// TIA Portal V16 export
// export: Created 2021-08-10T11:53:40.4139441Z, ExportSetting WithDefaults, WithReadOnly, DisplayName Totally Integrated Automation Portal, DisplayVersion V16, DisplayName TIA Portal Version Control Interface, DisplayVersion V16, DisplayName TIA Portal Openness, DisplayVersion V16, DisplayName TIA Portal Teamcenter Gateway, DisplayVersion V16, DisplayName SINAMICS Startdrive Advanced, DisplayVersion V16, DisplayName SINAMICS Startdrive G130, G150, S120, S150, SINAMICS MV, S210, DisplayVersion V16, DisplayName SINAMICS Startdrive G110M, G120, G120C, G120D, G120P, DisplayVersion V16, DisplayName STEP 7 Professional, DisplayVersion V16, DisplayName STEP 7 Safety, DisplayVersion V16, DisplayName WinCC Unified SCADA Engineering System, DisplayVersion V16
FUNCTION_BLOCK "fbValve_Solenoid"   // FB110, FBD
TITLE = Controls a double- or single-acting valve
{ S7_Optimized_Access := 'TRUE' }
VERSION : 0.1
// stored: AutoNumber false, CodeModifiedDate 2021-08-10T11:52:58.0273326Z, CompileDate 2021-08-10T11:53:23.0999729Z, CreationDate 2020-02-26T07:34:28.9567791Z, DownloadWithoutReinit false, HandleErrorsWithinBlock false, InterfaceModifiedDate 2019-07-17T06:42:37.7805928Z, IsConsistent true, IsIECCheckEnabled false, IsKnowHowProtected false, ISMultiInstanceCapable true, IsRetainMemResEnabled false, IsWriteProtected false, LibraryConformanceStatus Warning: The object contains access to global PLC constants., LibraryType fbValve_Solenoid V 3.0.6 in test, LibraryTypeVersionGuid 0a9fd967-cd2b-46e1-afc3-82055bb762c7, MemoryReserve 100, ModifiedDate 2021-08-10T11:52:58.0273326Z, ParameterModified 2019-07-17T06:42:37.7805928Z, PLCSimAdvancedSupport true, SetENOAutomatically false, StructureModified 2019-07-17T06:42:37.7805928Z, UDAEnableTagReadback false
   VAR_INPUT
      tInTimeout { ExternalAccessible := 'False'; ExternalVisible := 'False'; ExternalWritable := 'False'} : Time;   // Timeout time for an actuator's feedback to activate before giving a fault
      iInMode { ExternalAccessible := 'False'; ExternalVisible := 'False'; ExternalWritable := 'False'} : Int;   // Mode Selection
      bInEstop { ExternalAccessible := 'False'; ExternalVisible := 'False'; ExternalWritable := 'False'} : Bool;   // Estop
      bInSignalHome { ExternalAccessible := 'False'; ExternalVisible := 'False'; ExternalWritable := 'False'} : Bool;   // Home position feedback
      bInSignalWork { ExternalAccessible := 'False'; ExternalVisible := 'False'; ExternalWritable := 'False'} : Bool;   // Work position feedback
      bInEnable { ExternalAccessible := 'False'; ExternalVisible := 'False'; ExternalWritable := 'False'} : Bool;   // Home and Work Enabled
      bInCommandWork { ExternalAccessible := 'False'; ExternalVisible := 'False'; ExternalWritable := 'False'} : Bool;   // Move to work position in automatic mode
      bInResetError { ExternalAccessible := 'False'; ExternalVisible := 'False'; ExternalWritable := 'False'} : Bool;   // Reset Error
      bInSimulate { ExternalAccessible := 'False'; ExternalVisible := 'False'; ExternalWritable := 'False'} : Bool;   // Activate device simulation
   END_VAR
   VAR_OUTPUT
      bOutCommandHome { ExternalAccessible := 'False'; ExternalVisible := 'False'; ExternalWritable := 'False'} : Bool;   // Home position command
      bOutCommandWork { ExternalAccessible := 'False'; ExternalVisible := 'False'; ExternalWritable := 'False'} : Bool;   // Work position command
      bOutActiveHome { ExternalAccessible := 'False'; ExternalVisible := 'False'; ExternalWritable := 'False'} : Bool;   // Valve is in home position
      bOutActiveWork { ExternalAccessible := 'False'; ExternalVisible := 'False'; ExternalWritable := 'False'} : Bool;   // Valve is in work position
      bOutAuto { ExternalAccessible := 'False'; ExternalVisible := 'False'; ExternalWritable := 'False'} : Bool;   // Block in auto mode
      bOutError { ExternalAccessible := 'False'; ExternalVisible := 'False'; ExternalWritable := 'False'} : Bool;   // Error exists
      ERROR_Valve { ExternalAccessible := 'False'; ExternalVisible := 'False'; ExternalWritable := 'False'} : "udtError_Valve";   // Valve error structure
   END_VAR
   VAR_IN_OUT
      HMI_ValveControl : "udtHMI_ValveControl";   // HMI valve control
   END_VAR
   VAR
      ErrorScroller { ExternalAccessible := 'False'; ExternalVisible := 'False'; ExternalWritable := 'False'; S7_SetPoint := 'True'} : "fbErrorScroller";   // Sub-block to handle error scroller
      TON_TimeOut { ExternalAccessible := 'False'; ExternalVisible := 'False'; ExternalWritable := 'False'; S7_SetPoint := 'True'} : TON_TIME;   // Timer for Error Timeout
      iLastMode { ExternalAccessible := 'False'; ExternalVisible := 'False'; ExternalWritable := 'False'} : Int;   // Last mode code
      bNewMode { ExternalAccessible := 'False'; ExternalVisible := 'False'; ExternalWritable := 'False'} : Bool;   // New mode selected
      bEnableHome { ExternalAccessible := 'False'; ExternalVisible := 'False'; ExternalWritable := 'False'} : Bool;   // Home position enabled
      bEnableWork { ExternalAccessible := 'False'; ExternalVisible := 'False'; ExternalWritable := 'False'} : Bool;   // Work position enabled
      bAutoMode { ExternalAccessible := 'False'; ExternalVisible := 'False'; ExternalWritable := 'False'} : Bool;   // Auto Mode is active
      bManualMode { ExternalAccessible := 'False'; ExternalVisible := 'False'; ExternalWritable := 'False'} : Bool;   // Manual Mode is active
      bReset { ExternalAccessible := 'False'; ExternalVisible := 'False'; ExternalWritable := 'False'} : Bool;
      bTON_TimeOut { ExternalAccessible := 'False'; ExternalVisible := 'False'; ExternalWritable := 'False'} : Bool;
      bPB_Home { ExternalAccessible := 'False'; ExternalVisible := 'False'; ExternalWritable := 'False'} : Bool;
      bPB_Work { ExternalAccessible := 'False'; ExternalVisible := 'False'; ExternalWritable := 'False'} : Bool;
      bPB_ResetError { ExternalAccessible := 'False'; ExternalVisible := 'False'; ExternalWritable := 'False'} : Bool;
   END_VAR
   VAR_TEMP
      tTimeoutElapsed : Time;   // Elapsed time for TON_Timeout
      bTemp : Bool;
   END_VAR
   VAR_TEMP   // added for the SCL form of the ladder/FBD networks
      _w1 : Bool;
      _w2 : Bool;
   END_VAR
BEGIN

REGION Network 1: --------------------------------------------------------- Inputs ------------------------------------------------------------------
END_REGION

REGION Network 2: Read HMI input buttons
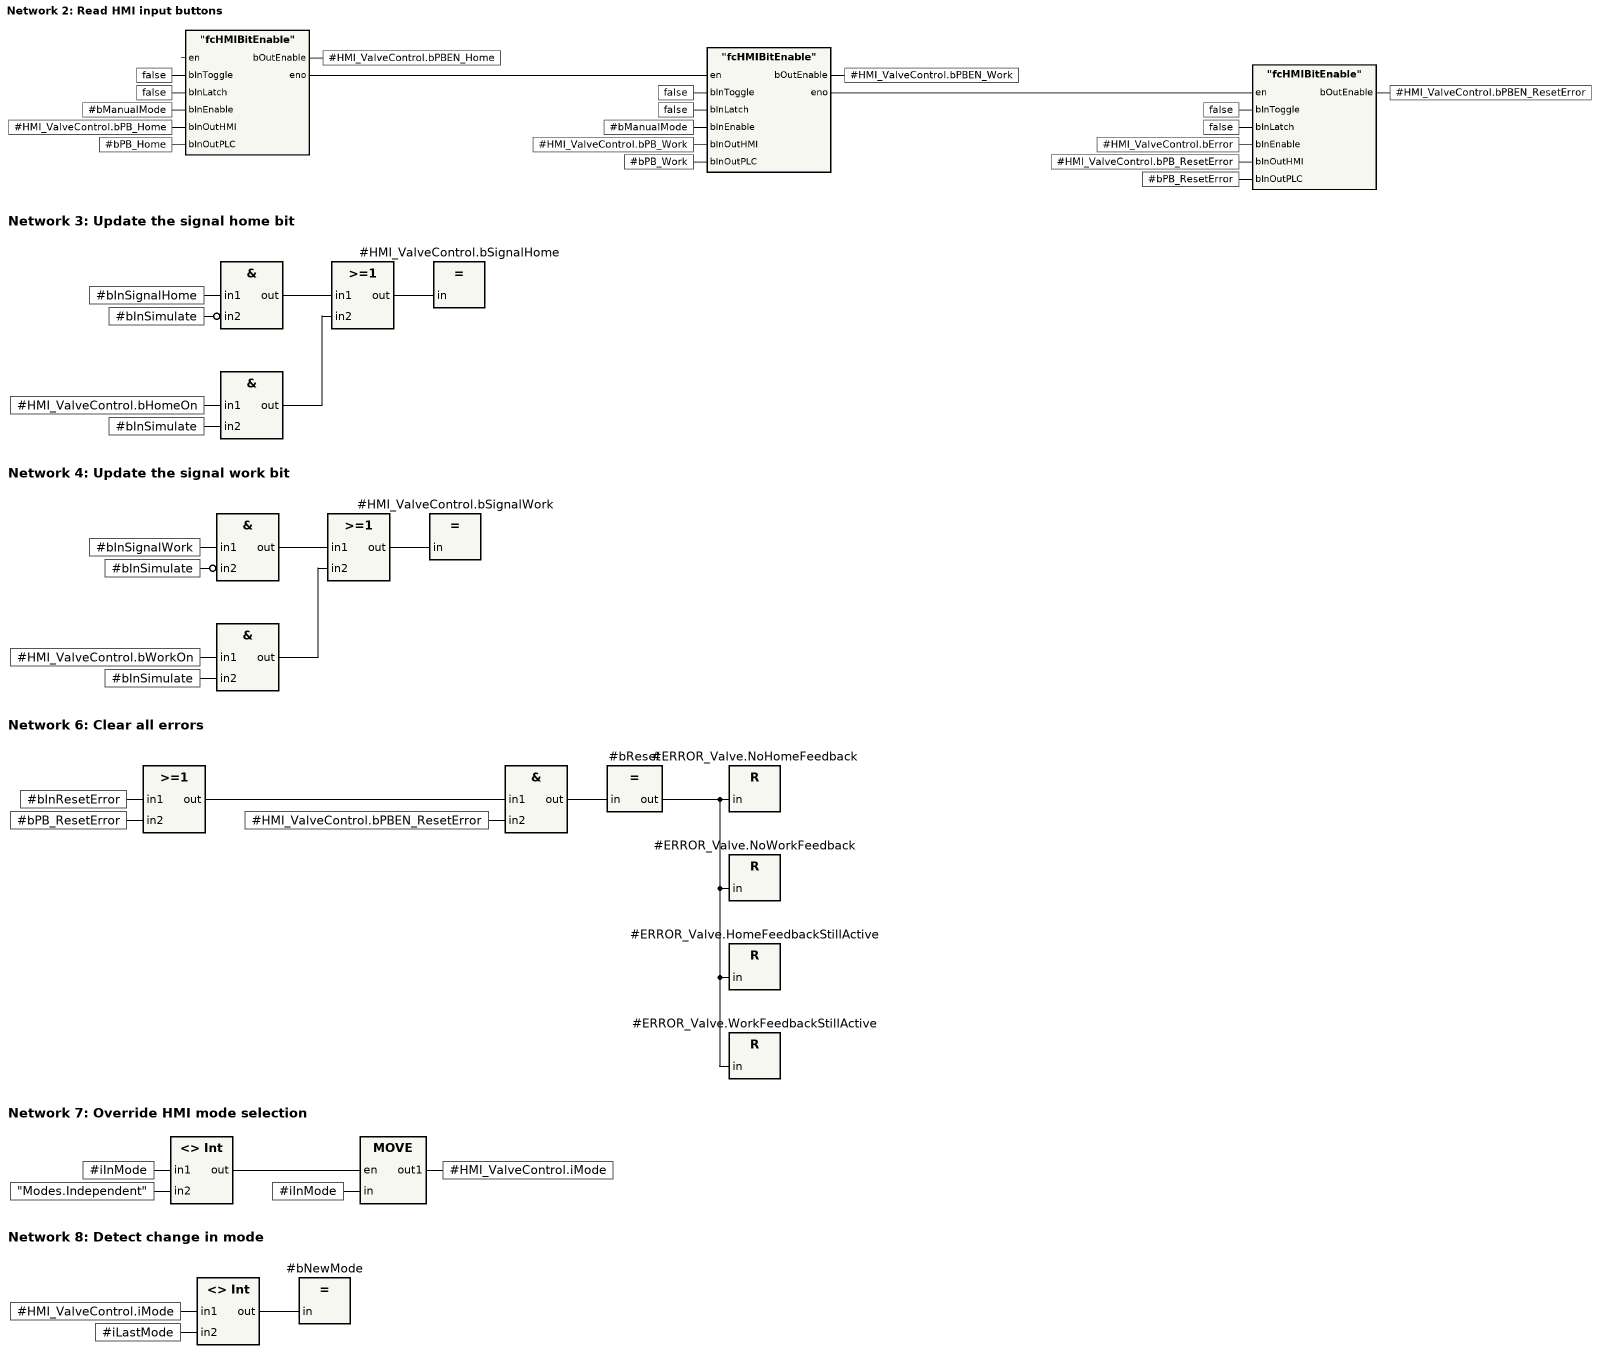
   "fcHMIBitEnable"(bInToggle := false,
                    bInLatch := false,
                    bInEnable := #bManualMode,
                    bInOutHMI := #HMI_ValveControl.bPB_Home,
                    bInOutPLC := #bPB_Home,
                    bOutEnable => #HMI_ValveControl.bPBEN_Home,
                    ENO => #_w1);
   "fcHMIBitEnable"(EN := #_w1,
                    bInToggle := false,
                    bInLatch := false,
                    bInEnable := #bManualMode,
                    bInOutHMI := #HMI_ValveControl.bPB_Work,
                    bInOutPLC := #bPB_Work,
                    bOutEnable => #HMI_ValveControl.bPBEN_Work,
                    ENO => #_w2);
   IF #_w2 THEN
       "fcHMIBitEnable"(bInToggle := false,
                        bInLatch := false,
                        bInEnable := #HMI_ValveControl.bError,
                        bInOutHMI := #HMI_ValveControl.bPB_ResetError,
                        bInOutPLC := #bPB_ResetError,
                        bOutEnable => #HMI_ValveControl.bPBEN_ResetError);
   END_IF;
END_REGION

REGION Network 3: Update the signal home bit
   #HMI_ValveControl.bSignalHome := (#bInSignalHome AND NOT #bInSimulate) OR (#HMI_ValveControl.bHomeOn AND #bInSimulate);
END_REGION

REGION Network 4: Update the signal work bit
   #HMI_ValveControl.bSignalWork := (#bInSignalWork AND NOT #bInSimulate) OR (#HMI_ValveControl.bWorkOn AND #bInSimulate);
END_REGION

REGION Network 5: --------------------------------------------------- Control Logic ------------------------------------------------------------
END_REGION

REGION Network 6: Clear all errors
   #bReset := (#bInResetError OR #bPB_ResetError) AND #HMI_ValveControl.bPBEN_ResetError;
   IF #bReset THEN
       #ERROR_Valve.NoHomeFeedback := FALSE;
       #ERROR_Valve.NoWorkFeedback := FALSE;
       #ERROR_Valve.HomeFeedbackStillActive := FALSE;
       #ERROR_Valve.WorkFeedbackStillActive := FALSE;
   END_IF;
END_REGION

REGION Network 7: Override HMI mode selection
   IF #iInMode <> "Modes.Independent" THEN #HMI_ValveControl.iMode := #iInMode; END_IF;
END_REGION

REGION Network 8: Detect change in mode
   #bNewMode := #HMI_ValveControl.iMode <> #iLastMode;
END_REGION

REGION Network 9: Keep track of last mode
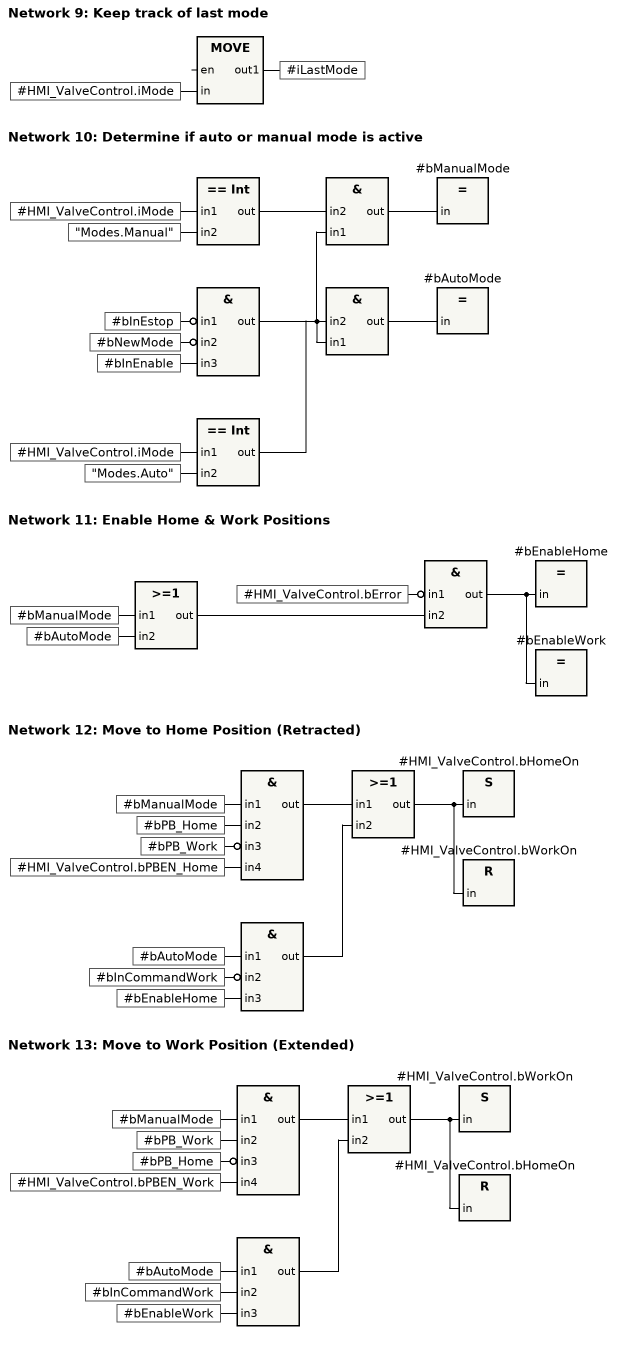
   #iLastMode := #HMI_ValveControl.iMode;
END_REGION

REGION Network 10: Determine if auto or manual mode is active
   #_w1 := NOT #bInEstop AND NOT #bNewMode AND #bInEnable;
   #bManualMode := (#HMI_ValveControl.iMode = "Modes.Manual") AND #_w1;
   #bAutoMode := (#HMI_ValveControl.iMode = "Modes.Auto") AND #_w1;
END_REGION

REGION Network 11: Enable Home & Work Positions
   // IF manual mode AND no estop AND not a new mode AND enabled => 
   // --if no cylinder errors, enable move to Home and Work
   // --enable home and work HMI buttons only in manual mode
   #bEnableHome := NOT #HMI_ValveControl.bError AND (#bManualMode OR #bAutoMode);
   #bEnableWork := #bEnableHome;
END_REGION

REGION Network 12: Move to Home Position (Retracted)
   // IF manual mode and home button is pressed =>
   // --Set close cylinder
   IF (#bManualMode AND #bPB_Home AND NOT #bPB_Work AND #HMI_ValveControl.bPBEN_Home) OR (#bAutoMode AND NOT #bInCommandWork AND #bEnableHome) THEN
       #HMI_ValveControl.bHomeOn := TRUE;
       #HMI_ValveControl.bWorkOn := FALSE;
   END_IF;
END_REGION

REGION Network 13: Move to Work Position (Extended)
   // IF manual mode and work button button is pressed =>
   // --Set open cylinder
   IF (#bManualMode AND #bPB_Work AND NOT #bPB_Home AND #HMI_ValveControl.bPBEN_Work) OR (#bAutoMode AND #bInCommandWork AND #bEnableWork) THEN
       #HMI_ValveControl.bWorkOn := TRUE;
       #HMI_ValveControl.bHomeOn := FALSE;
   END_IF;
END_REGION

REGION Network 14: Reset home on if not enabled
   // IF in auto AND home is not enabled => RESET home command
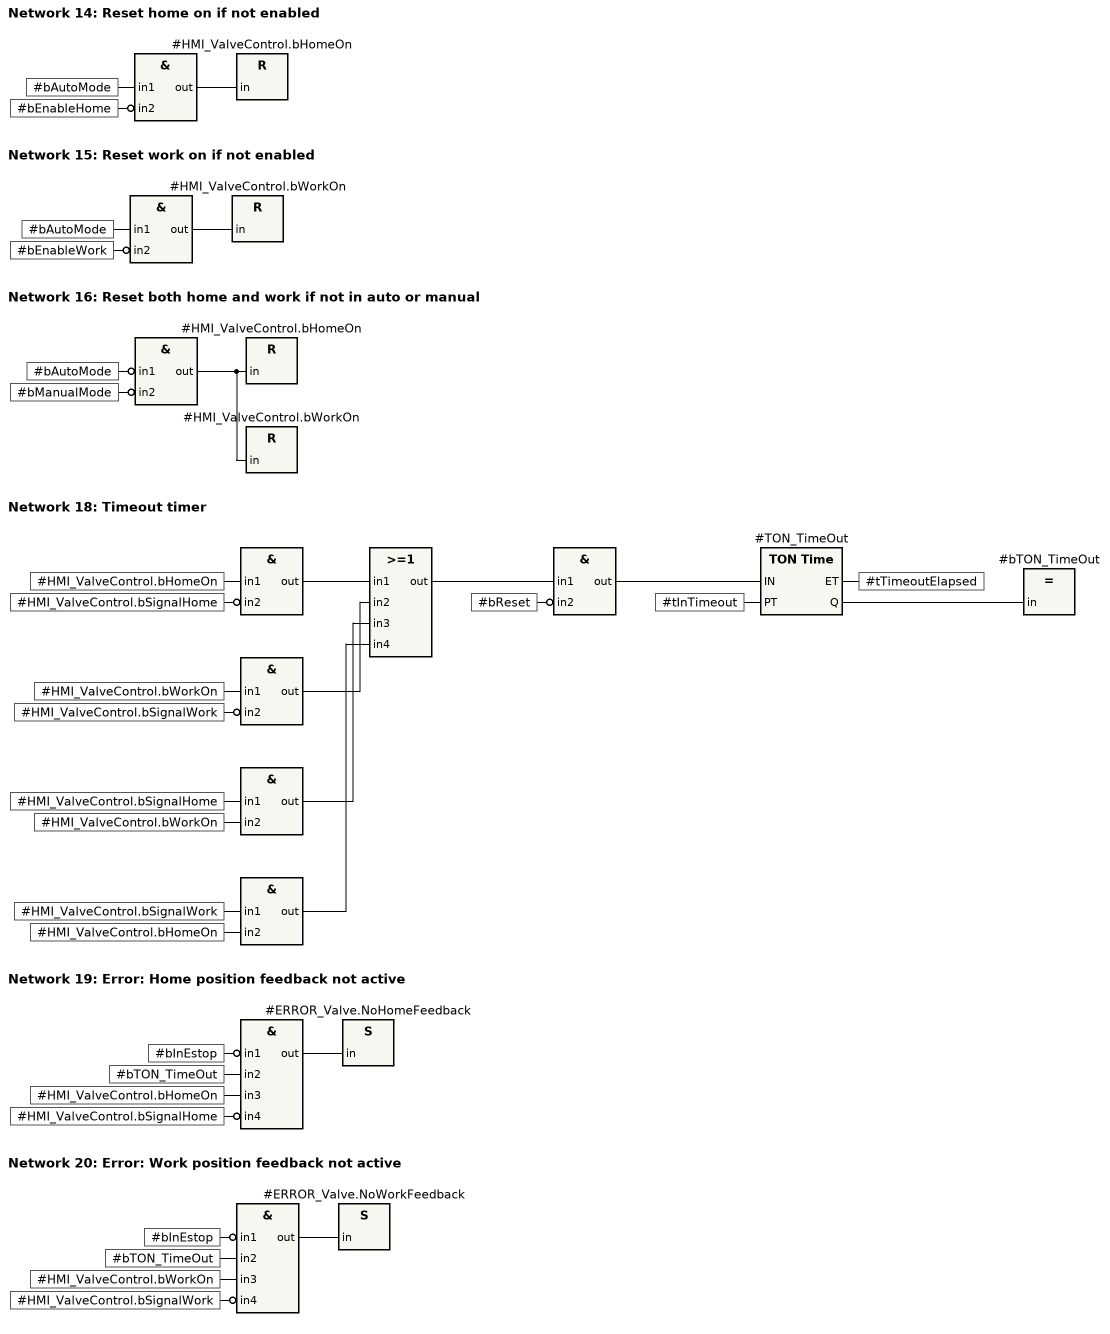
   IF #bAutoMode AND NOT #bEnableHome THEN #HMI_ValveControl.bHomeOn := FALSE; END_IF;
END_REGION

REGION Network 15: Reset work on if not enabled
   // IF in auto AND work is not enabled => RESET work command
   IF #bAutoMode AND NOT #bEnableWork THEN #HMI_ValveControl.bWorkOn := FALSE; END_IF;
END_REGION

REGION Network 16: Reset both home and work if not in auto or manual
   // IF not in auto AND not in manual => RESET home and work commands
   IF NOT #bAutoMode AND NOT #bManualMode THEN
       #HMI_ValveControl.bHomeOn := FALSE;
       #HMI_ValveControl.bWorkOn := FALSE;
   END_IF;
END_REGION

REGION Network 17: --------------------------------------------------------- Errors ------------------------------------------------------------------
END_REGION

REGION Network 18: Timeout timer
   // Time delay for errors
   #TON_TimeOut(IN := ((#HMI_ValveControl.bHomeOn AND NOT #HMI_ValveControl.bSignalHome) OR (#HMI_ValveControl.bWorkOn AND NOT #HMI_ValveControl.bSignalWork) OR (#HMI_ValveControl.bSignalHome AND #HMI_ValveControl.bWorkOn) OR (#HMI_ValveControl.bSignalWork AND #HMI_ValveControl.bHomeOn)) AND NOT #bReset,   // TON
                PT := #tInTimeout,
                ET => #tTimeoutElapsed);
   #bTON_TimeOut := #TON_TimeOut.Q;
END_REGION

REGION Network 19: Error: Home position feedback not active
   IF NOT #bInEstop AND #bTON_TimeOut AND #HMI_ValveControl.bHomeOn AND NOT #HMI_ValveControl.bSignalHome THEN
       #ERROR_Valve.NoHomeFeedback := TRUE;
   END_IF;
END_REGION

REGION Network 20: Error: Work position feedback not active
   // Not reach work position
   IF NOT #bInEstop AND #bTON_TimeOut AND #HMI_ValveControl.bWorkOn AND NOT #HMI_ValveControl.bSignalWork THEN
       #ERROR_Valve.NoWorkFeedback := TRUE;
   END_IF;
END_REGION

REGION Network 21: Error: Home position feedback still active
   // Home position still active
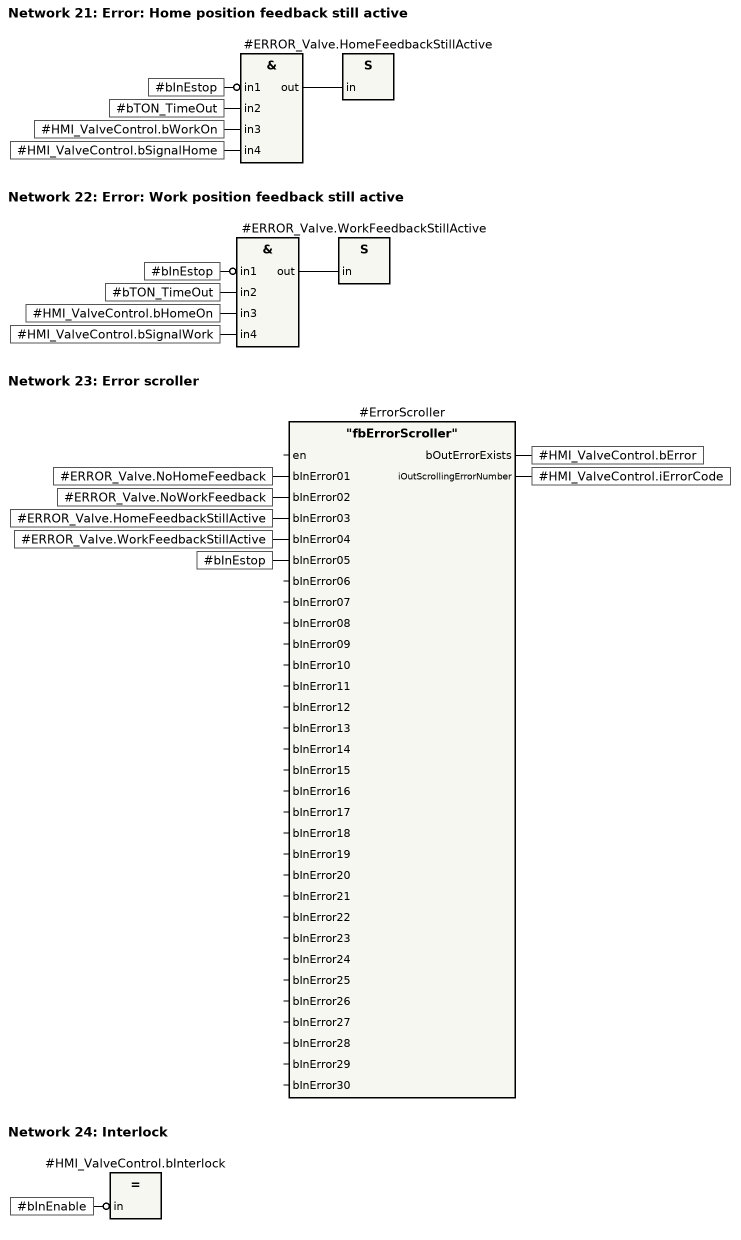
   IF NOT #bInEstop AND #bTON_TimeOut AND #HMI_ValveControl.bWorkOn AND #HMI_ValveControl.bSignalHome THEN
       #ERROR_Valve.HomeFeedbackStillActive := TRUE;
   END_IF;
END_REGION

REGION Network 22: Error: Work position feedback still active
   // Work position still active
   IF NOT #bInEstop AND #bTON_TimeOut AND #HMI_ValveControl.bHomeOn AND #HMI_ValveControl.bSignalWork THEN
       #ERROR_Valve.WorkFeedbackStillActive := TRUE;
   END_IF;
END_REGION

REGION Network 23: Error scroller
   // Call the Error-Scroller which cyles through all possible errors and checks 
   // their state for display on the HMI
   #ErrorScroller(bInError01 := #ERROR_Valve.NoHomeFeedback,   // "fbErrorScroller"
                  bInError02 := #ERROR_Valve.NoWorkFeedback,
                  bInError03 := #ERROR_Valve.HomeFeedbackStillActive,
                  bInError04 := #ERROR_Valve.WorkFeedbackStillActive,
                  bInError05 := #bInEstop,
                  bOutErrorExists => #HMI_ValveControl.bError,
                  iOutScrollingErrorNumber => #HMI_ValveControl.iErrorCode);
END_REGION

REGION Network 24: Interlock
   #HMI_ValveControl.bInterlock := NOT #bInEnable;
END_REGION

REGION Network 25: Set HMI status
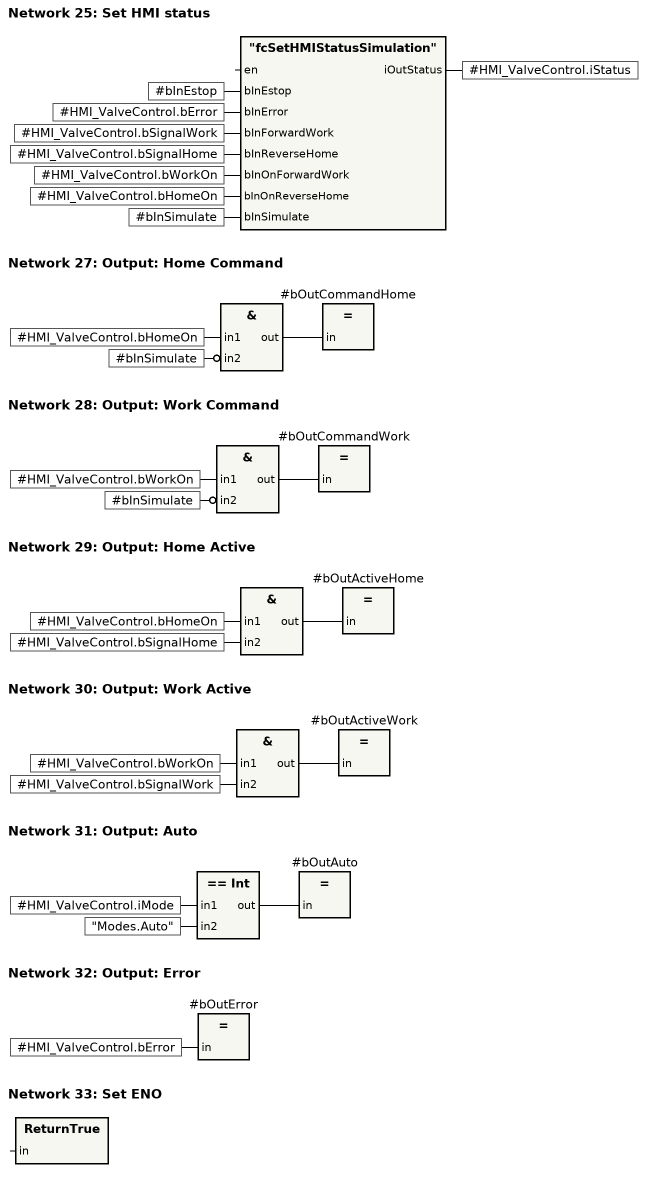
   "fcSetHMIStatusSimulation"(bInEstop := #bInEstop,
                           bInError := #HMI_ValveControl.bError,
                           bInForwardWork := #HMI_ValveControl.bSignalWork,
                           bInReverseHome := #HMI_ValveControl.bSignalHome,
                           bInOnForwardWork := #HMI_ValveControl.bWorkOn,
                           bInOnReverseHome := #HMI_ValveControl.bHomeOn,
                           bInSimulate := #bInSimulate,
                           iOutStatus => #HMI_ValveControl.iStatus);
END_REGION

REGION Network 26: -------------------------------------------------- Outputs --------------------------------------------------
END_REGION

REGION Network 27: Output: Home Command
   #bOutCommandHome := #HMI_ValveControl.bHomeOn AND NOT #bInSimulate;
END_REGION

REGION Network 28: Output: Work Command
   #bOutCommandWork := #HMI_ValveControl.bWorkOn AND NOT #bInSimulate;
END_REGION

REGION Network 29: Output: Home Active
   #bOutActiveHome := #HMI_ValveControl.bHomeOn AND #HMI_ValveControl.bSignalHome;
END_REGION

REGION Network 30: Output: Work Active
   #bOutActiveWork := #HMI_ValveControl.bWorkOn AND #HMI_ValveControl.bSignalWork;
END_REGION

REGION Network 31: Output: Auto
   #bOutAuto := #HMI_ValveControl.iMode = "Modes.Auto";
END_REGION

REGION Network 32: Output: Error
   #bOutError := #HMI_ValveControl.bError;
END_REGION

REGION Network 33: Set ENO
   ENO := TRUE;
   RETURN;
END_REGION
END_FUNCTION_BLOCK
